{attribute addProperty BoxType "EM7004-0000-9996"}
{attribute addProperty Id "PLS_EnabledAT %I*BOOL811Unequal_SI_0AT %I*BOOL812"}
{attribute addProperty CRC "557741559"}
{attribute addProperty SizeInBites "16"}
{attribute addProperty SizeInBytes "2"}
TYPE PLS_Inputs_213E75F7 :
STRUCT
	{attribute addProperty Name "PLS_Enabled"}
	PLS_Enabled AT %I* : BOOL;
	{attribute addProperty Name "Unequal_SI_0"}
	Unequal_SI_0 AT %I* : BOOL;
END_STRUCT
END_TYPE

(* stored: Version 1.2.0.0, ProductVersion 3.1.4024.9
   DUT PLS_Inputs_213E75F7: Id {5785c025-0478-4ded-b6a2-511f561da4d6} *)
